{attribute 'GeneratedUsingTerminal: EL3423-0000-0016'}
{attribute addProperty BoxType "EL3423-0000-0016"}
{attribute addProperty Id "Active_EnergyAT %I*LINT8Active_Positive_EnergyAT %I*ULINT8Active_Negative_EnergyAT %I*ULINT8"}
{attribute addProperty CRC "3383139009"}
{attribute addProperty Size "24"}
TYPE Total_Active_C9A69AC1 EXTENDS InputBase_8311D824 :
STRUCT
	{attribute addProperty Name "Active_Energy"}
	Active_Energy AT %I* : LINT;
	{attribute addProperty Name "Active_Positive_Energy"}
	Active_Positive_Energy AT %I* : ULINT;
	{attribute addProperty Name "Active_Negative_Energy"}
	Active_Negative_Energy AT %I* : ULINT;
END_STRUCT
END_TYPE

(* stored: Version 1.2.0.0, ProductVersion 3.1.4024.11
   DUT Total_Active_C9A69AC1: Id {6d004799-5945-42f1-82f9-39a93cc39196} *)
